// TIA Portal V16 export
// export: Created 2021-11-12T13:32:46.6984592Z, ExportSetting WithDefaults, DisplayName Totally Integrated Automation Portal, DisplayVersion V16 Update 3, DisplayName TIA Portal Version Control Interface, DisplayVersion V16 Update 2, DisplayName TIA Portal Openness, DisplayVersion V16 Update 3, DisplayName SINAMICS Startdrive Advanced, DisplayVersion V16 Update 5, DisplayName SINAMICS Startdrive G130, G150, S120, S150, SINAMICS MV, S210, DisplayVersion V16 Update 5, DisplayName SINAMICS Startdrive G110M, G120, G120C, G120D, G120P, G115D, DisplayVersion V16 Update 5, DisplayName STEP 7 Professional, DisplayVersion V16 Update 3, DisplayName STEP 7 Safety, DisplayVersion V16, DisplayName WinCC UA Professional, DisplayVersion V16 Update 3
DATA_BLOCK "IDB_Zone200"   // DB26
VERSION : 0.1
// stored: AutoNumber true, DBAccessibleFromOPCUA true, InstanceOfName Zone200, InstanceOfType FB
"Zone200"
   // VAR
   //    SF_ZoneMode { S7_SetPoint := 'True'} : "STD_Zone";
   //    SF_Station210Mode { S7_SetPoint := 'True'} : "STD_Station";
   //    SF_Station220Mode { S7_SetPoint := 'True'} : "STD_Station";
   //    SF_Station230Mode { S7_SetPoint := 'True'} : "STD_Station";
   //    SF_Station2R1Mode { S7_SetPoint := 'True'} : "STD_Station";
   //    SF_Station2R2Mode { S7_SetPoint := 'True'} : "STD_Station";
   //    SF_StationSCH1Mode { S7_SetPoint := 'True'} : "STD_Station";
   //    SF_StationBSN3Mode { S7_SetPoint := 'True'} : "STD_Station";
   //    SF_CameraLights { S7_SetPoint := 'True'} : "STD_OnOff";
   //    SS_Edge { S7_SetPoint := 'True'} : Array[0..100] of Bool;
   //    SB1CameraLightsON { S7_SetPoint := 'True'} : Bool;
   // END_VAR
BEGIN
END_DATA_BLOCK
